// LS Electric XG5000 project: baraka_plc
// PLC NewPLC
// module base 0 slot 0: Input/Output Module:XBC-DR10E (DC 24V INPUT 6points/RELAY OUTPUT 4points)

PROGRAM Program (task: Scan Program)

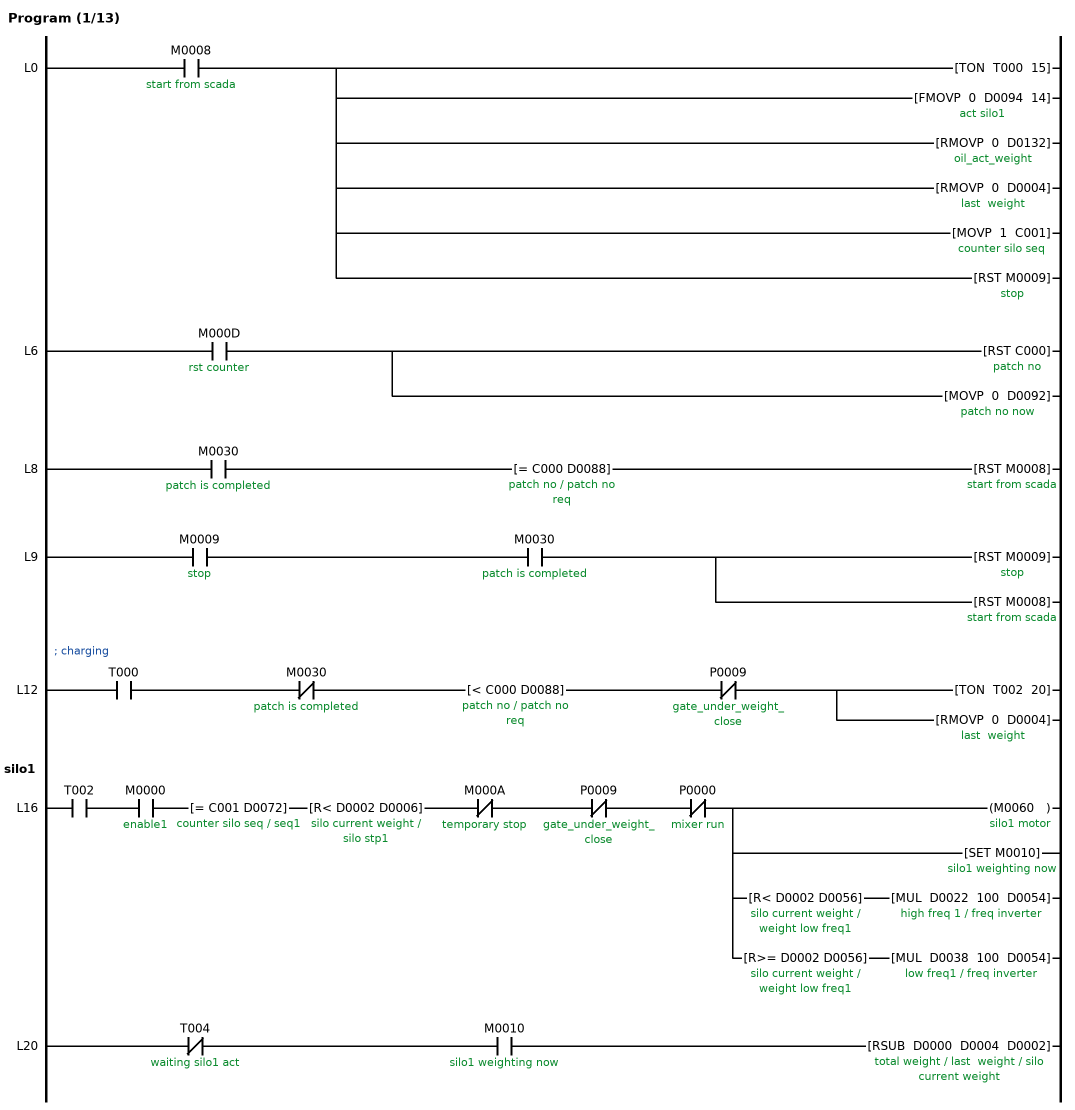
; L0
LOAD      M0008	// start from scada
TON       T000 15
FMOVP     0 D0094 14	// act silo1
RMOVP     0 D0132	// oil_act_weight
RMOVP     0 D0004	// last  weight
MOVP      1 C001	// counter silo seq
RST       M0009	// stop
; L6
LOAD      M000D	// rst counter
RST       C000	// patch no
MOVP      0 D0092	// patch no now
; L8
LOAD      M0030	// patch is completed
AND=      C000 D0088	// patch no / patch no req
RST       M0008	// start from scada
; L9
LOAD      M0009	// stop
AND       M0030	// patch is completed
RST       M0009	// stop
RST       M0008	// start from scada
// charging
; L12
LOAD      T000
AND NOT   M0030	// patch is completed
AND<      C000 D0088	// patch no / patch no req
AND NOT   P0009	// gate_under_weight_close
TON       T002 20
RMOVP     0 D0004	// last  weight
silo1:
; L16
LOAD      T002
AND       M0000	// enable1
AND=      C001 D0072	// counter silo seq / seq1
ANDR<     D0002 D0006	// silo current weight / silo stp1
AND NOT   M000A	// temporary stop
AND NOT   P0009	// gate_under_weight_close
AND NOT   P0000	// mixer run
OUT       M0060	// silo1 motor
SET       M0010	// silo1 weighting now
MPUSH
ANDR<     D0002 D0056	// silo current weight / weight low freq1
MUL       D0022 100 D0054	// high freq 1 / freq inverter
MPOP
ANDR>=    D0002 D0056	// silo current weight / weight low freq1
MUL       D0038 100 D0054	// low freq1 / freq inverter
; L20
LOAD NOT  T004	// waiting silo1 act
AND       M0010	// silo1 weighting now
RSUB      D0000 D0004 D0002	// total weight / last  weight / silo current weight

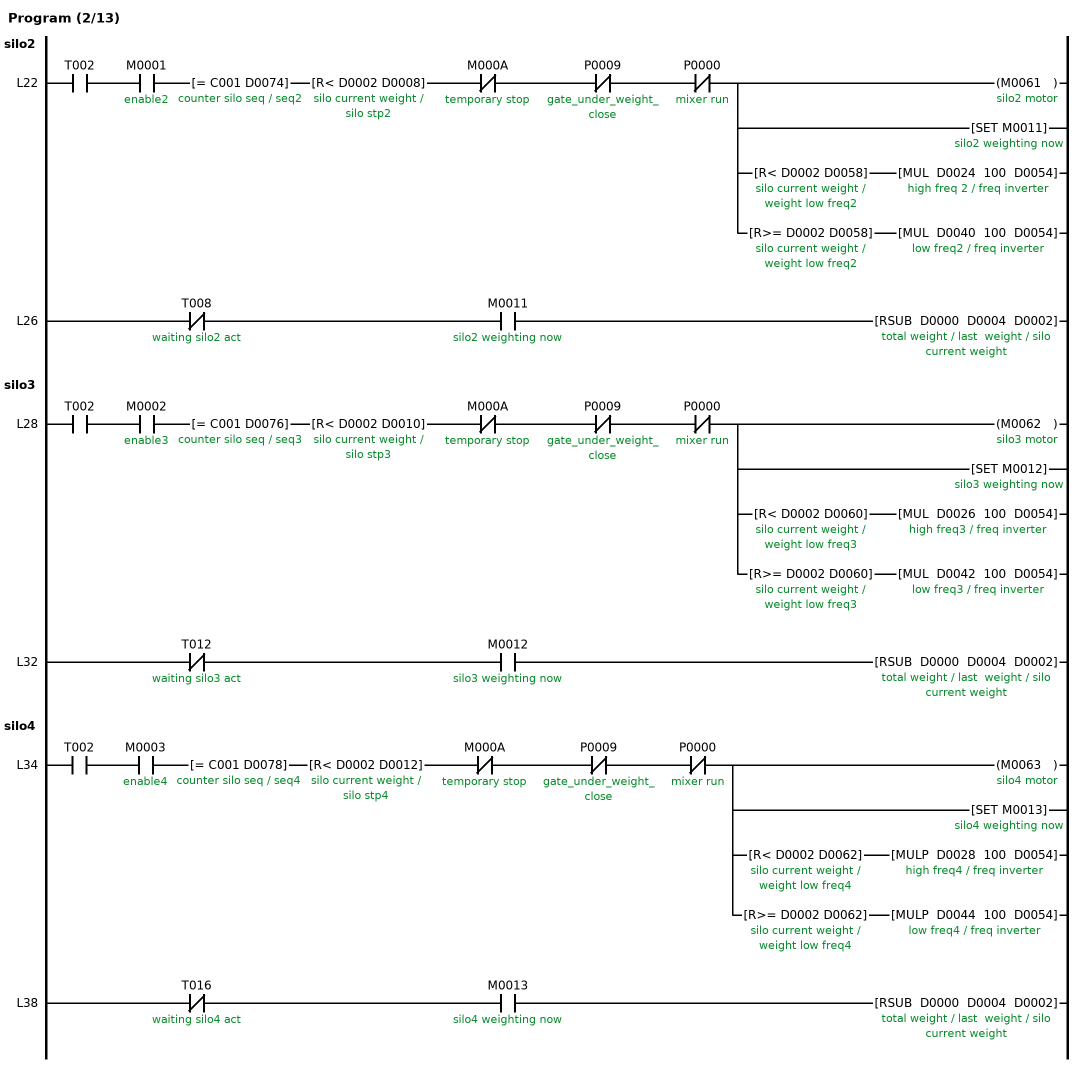
silo2:
; L22
LOAD      T002
AND       M0001	// enable2
AND=      C001 D0074	// counter silo seq / seq2
ANDR<     D0002 D0008	// silo current weight / silo stp2
AND NOT   M000A	// temporary stop
AND NOT   P0009	// gate_under_weight_close
AND NOT   P0000	// mixer run
OUT       M0061	// silo2 motor
SET       M0011	// silo2 weighting now
MPUSH
ANDR<     D0002 D0058	// silo current weight / weight low freq2
MUL       D0024 100 D0054	// high freq 2 / freq inverter
MPOP
ANDR>=    D0002 D0058	// silo current weight / weight low freq2
MUL       D0040 100 D0054	// low freq2 / freq inverter
; L26
LOAD NOT  T008	// waiting silo2 act
AND       M0011	// silo2 weighting now
RSUB      D0000 D0004 D0002	// total weight / last  weight / silo current weight
silo3:
; L28
LOAD      T002
AND       M0002	// enable3
AND=      C001 D0076	// counter silo seq / seq3
ANDR<     D0002 D0010	// silo current weight / silo stp3
AND NOT   M000A	// temporary stop
AND NOT   P0009	// gate_under_weight_close
AND NOT   P0000	// mixer run
OUT       M0062	// silo3 motor
SET       M0012	// silo3 weighting now
MPUSH
ANDR<     D0002 D0060	// silo current weight / weight low freq3
MUL       D0026 100 D0054	// high freq3 / freq inverter
MPOP
ANDR>=    D0002 D0060	// silo current weight / weight low freq3
MUL       D0042 100 D0054	// low freq3 / freq inverter
; L32
LOAD NOT  T012	// waiting silo3 act
AND       M0012	// silo3 weighting now
RSUB      D0000 D0004 D0002	// total weight / last  weight / silo current weight
silo4:
; L34
LOAD      T002
AND       M0003	// enable4
AND=      C001 D0078	// counter silo seq / seq4
ANDR<     D0002 D0012	// silo current weight / silo stp4
AND NOT   M000A	// temporary stop
AND NOT   P0009	// gate_under_weight_close
AND NOT   P0000	// mixer run
OUT       M0063	// silo4 motor
SET       M0013	// silo4 weighting now
MPUSH
ANDR<     D0002 D0062	// silo current weight / weight low freq4
MULP      D0028 100 D0054	// high freq4 / freq inverter
MPOP
ANDR>=    D0002 D0062	// silo current weight / weight low freq4
MULP      D0044 100 D0054	// low freq4 / freq inverter
; L38
LOAD NOT  T016	// waiting silo4 act
AND       M0013	// silo4 weighting now
RSUB      D0000 D0004 D0002	// total weight / last  weight / silo current weight

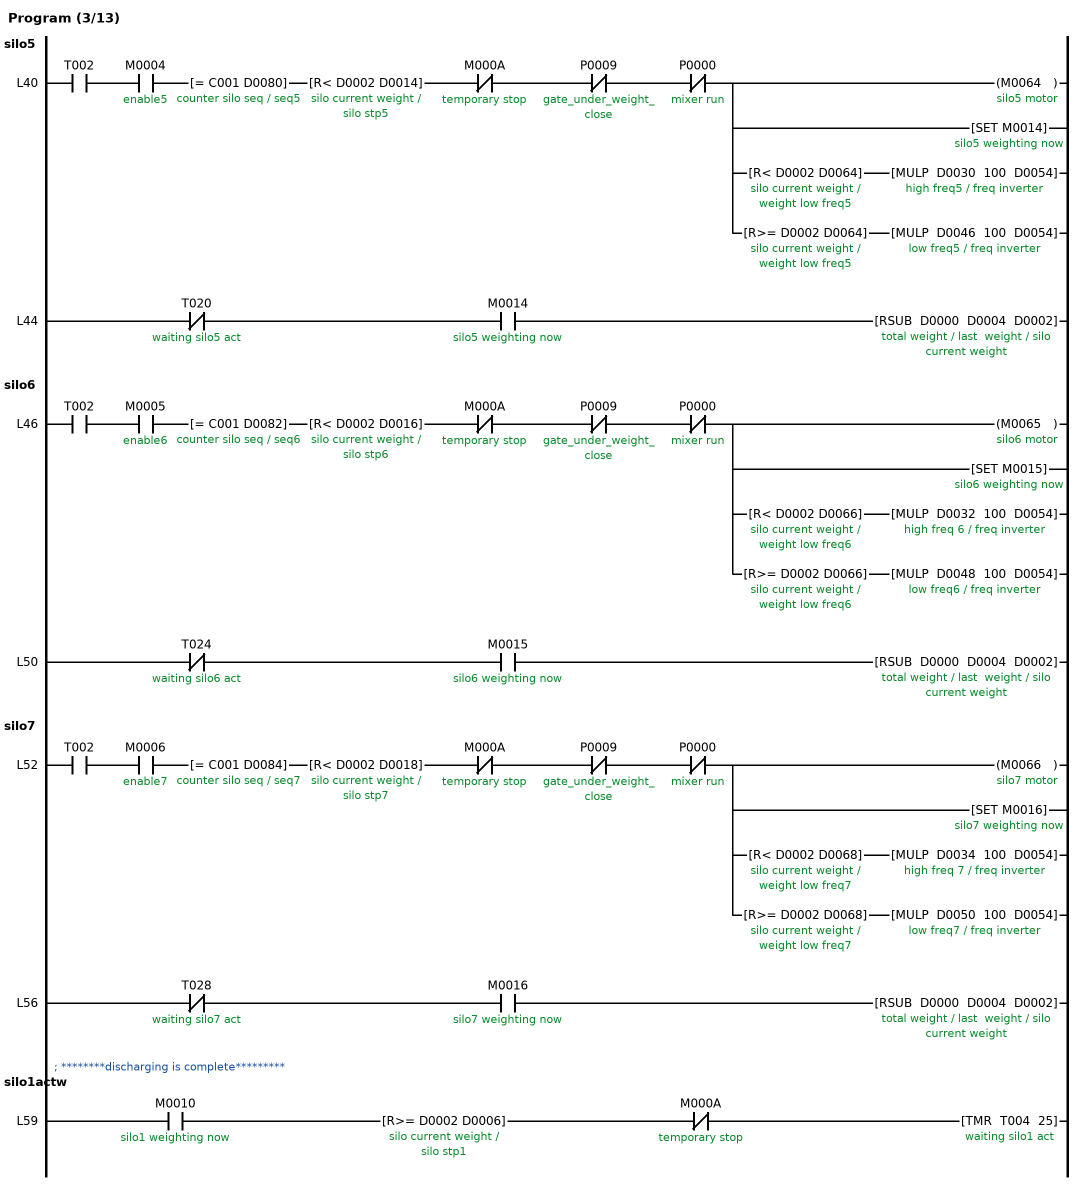
silo5:
; L40
LOAD      T002
AND       M0004	// enable5
AND=      C001 D0080	// counter silo seq / seq5
ANDR<     D0002 D0014	// silo current weight / silo stp5
AND NOT   M000A	// temporary stop
AND NOT   P0009	// gate_under_weight_close
AND NOT   P0000	// mixer run
OUT       M0064	// silo5 motor
SET       M0014	// silo5 weighting now
MPUSH
ANDR<     D0002 D0064	// silo current weight / weight low freq5
MULP      D0030 100 D0054	// high freq5 / freq inverter
MPOP
ANDR>=    D0002 D0064	// silo current weight / weight low freq5
MULP      D0046 100 D0054	// low freq5 / freq inverter
; L44
LOAD NOT  T020	// waiting silo5 act
AND       M0014	// silo5 weighting now
RSUB      D0000 D0004 D0002	// total weight / last  weight / silo current weight
silo6:
; L46
LOAD      T002
AND       M0005	// enable6
AND=      C001 D0082	// counter silo seq / seq6
ANDR<     D0002 D0016	// silo current weight / silo stp6
AND NOT   M000A	// temporary stop
AND NOT   P0009	// gate_under_weight_close
AND NOT   P0000	// mixer run
OUT       M0065	// silo6 motor
SET       M0015	// silo6 weighting now
MPUSH
ANDR<     D0002 D0066	// silo current weight / weight low freq6
MULP      D0032 100 D0054	// high freq 6 / freq inverter
MPOP
ANDR>=    D0002 D0066	// silo current weight / weight low freq6
MULP      D0048 100 D0054	// low freq6 / freq inverter
; L50
LOAD NOT  T024	// waiting silo6 act
AND       M0015	// silo6 weighting now
RSUB      D0000 D0004 D0002	// total weight / last  weight / silo current weight
silo7:
; L52
LOAD      T002
AND       M0006	// enable7
AND=      C001 D0084	// counter silo seq / seq7
ANDR<     D0002 D0018	// silo current weight / silo stp7
AND NOT   M000A	// temporary stop
AND NOT   P0009	// gate_under_weight_close
AND NOT   P0000	// mixer run
OUT       M0066	// silo7 motor
SET       M0016	// silo7 weighting now
MPUSH
ANDR<     D0002 D0068	// silo current weight / weight low freq7
MULP      D0034 100 D0054	// high freq 7 / freq inverter
MPOP
ANDR>=    D0002 D0068	// silo current weight / weight low freq7
MULP      D0050 100 D0054	// low freq7 / freq inverter
; L56
LOAD NOT  T028	// waiting silo7 act
AND       M0016	// silo7 weighting now
RSUB      D0000 D0004 D0002	// total weight / last  weight / silo current weight
// ********discharging is complete*********
silo1actw:
; L59
LOAD      M0010	// silo1 weighting now
ANDR>=    D0002 D0006	// silo current weight / silo stp1
AND NOT   M000A	// temporary stop
TMR       T004 25	// waiting silo1 act

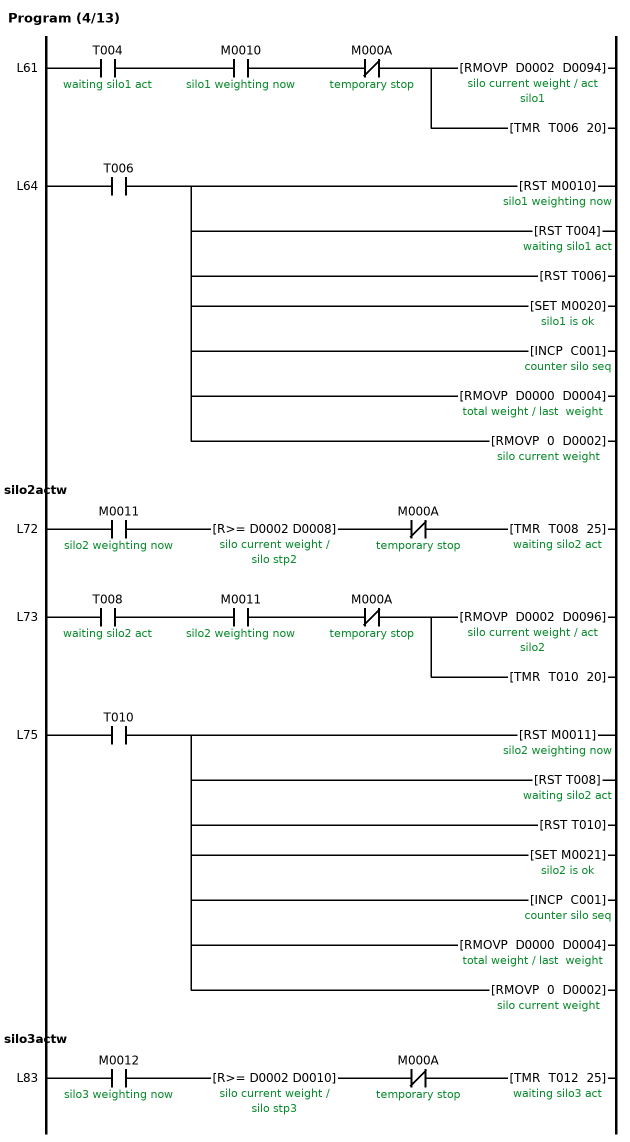
; L61
LOAD      T004	// waiting silo1 act
AND       M0010	// silo1 weighting now
AND NOT   M000A	// temporary stop
RMOVP     D0002 D0094	// silo current weight / act silo1
TMR       T006 20
; L64
LOAD      T006
RST       M0010	// silo1 weighting now
RST       T004	// waiting silo1 act
RST       T006
SET       M0020	// silo1 is ok
INCP      C001	// counter silo seq
RMOVP     D0000 D0004	// total weight / last  weight
RMOVP     0 D0002	// silo current weight
silo2actw:
; L72
LOAD      M0011	// silo2 weighting now
ANDR>=    D0002 D0008	// silo current weight / silo stp2
AND NOT   M000A	// temporary stop
TMR       T008 25	// waiting silo2 act
; L73
LOAD      T008	// waiting silo2 act
AND       M0011	// silo2 weighting now
AND NOT   M000A	// temporary stop
RMOVP     D0002 D0096	// silo current weight / act silo2
TMR       T010 20
; L75
LOAD      T010
RST       M0011	// silo2 weighting now
RST       T008	// waiting silo2 act
RST       T010
SET       M0021	// silo2 is ok
INCP      C001	// counter silo seq
RMOVP     D0000 D0004	// total weight / last  weight
RMOVP     0 D0002	// silo current weight
silo3actw:
; L83
LOAD      M0012	// silo3 weighting now
ANDR>=    D0002 D0010	// silo current weight / silo stp3
AND NOT   M000A	// temporary stop
TMR       T012 25	// waiting silo3 act

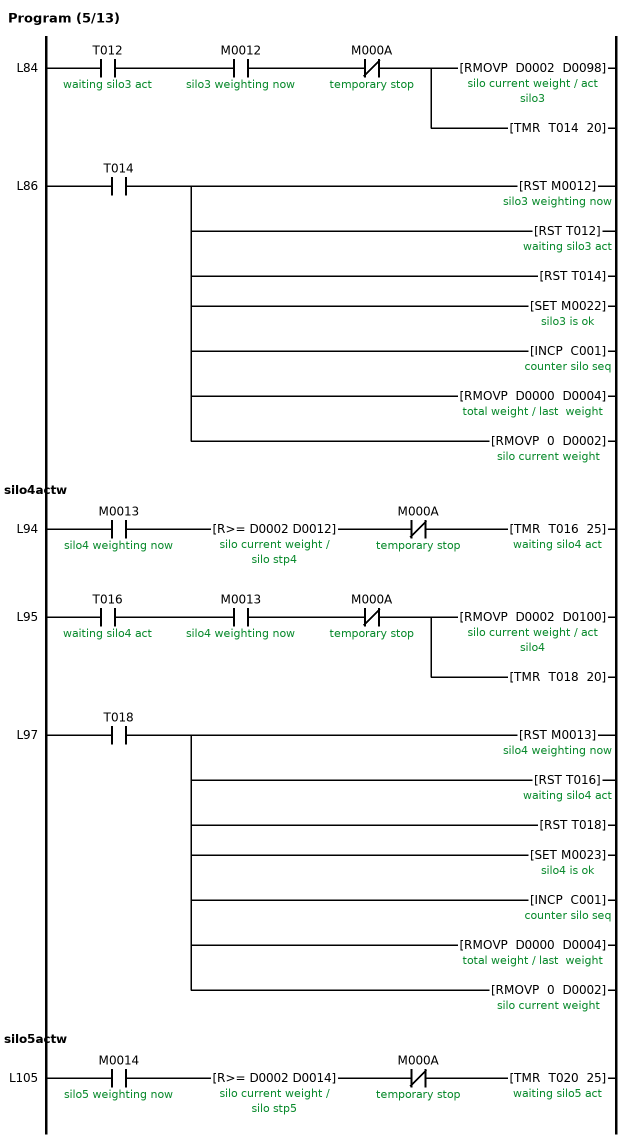
; L84
LOAD      T012	// waiting silo3 act
AND       M0012	// silo3 weighting now
AND NOT   M000A	// temporary stop
RMOVP     D0002 D0098	// silo current weight / act silo3
TMR       T014 20
; L86
LOAD      T014
RST       M0012	// silo3 weighting now
RST       T012	// waiting silo3 act
RST       T014
SET       M0022	// silo3 is ok
INCP      C001	// counter silo seq
RMOVP     D0000 D0004	// total weight / last  weight
RMOVP     0 D0002	// silo current weight
silo4actw:
; L94
LOAD      M0013	// silo4 weighting now
ANDR>=    D0002 D0012	// silo current weight / silo stp4
AND NOT   M000A	// temporary stop
TMR       T016 25	// waiting silo4 act
; L95
LOAD      T016	// waiting silo4 act
AND       M0013	// silo4 weighting now
AND NOT   M000A	// temporary stop
RMOVP     D0002 D0100	// silo current weight / act silo4
TMR       T018 20
; L97
LOAD      T018
RST       M0013	// silo4 weighting now
RST       T016	// waiting silo4 act
RST       T018
SET       M0023	// silo4 is ok
INCP      C001	// counter silo seq
RMOVP     D0000 D0004	// total weight / last  weight
RMOVP     0 D0002	// silo current weight
silo5actw:
; L105
LOAD      M0014	// silo5 weighting now
ANDR>=    D0002 D0014	// silo current weight / silo stp5
AND NOT   M000A	// temporary stop
TMR       T020 25	// waiting silo5 act

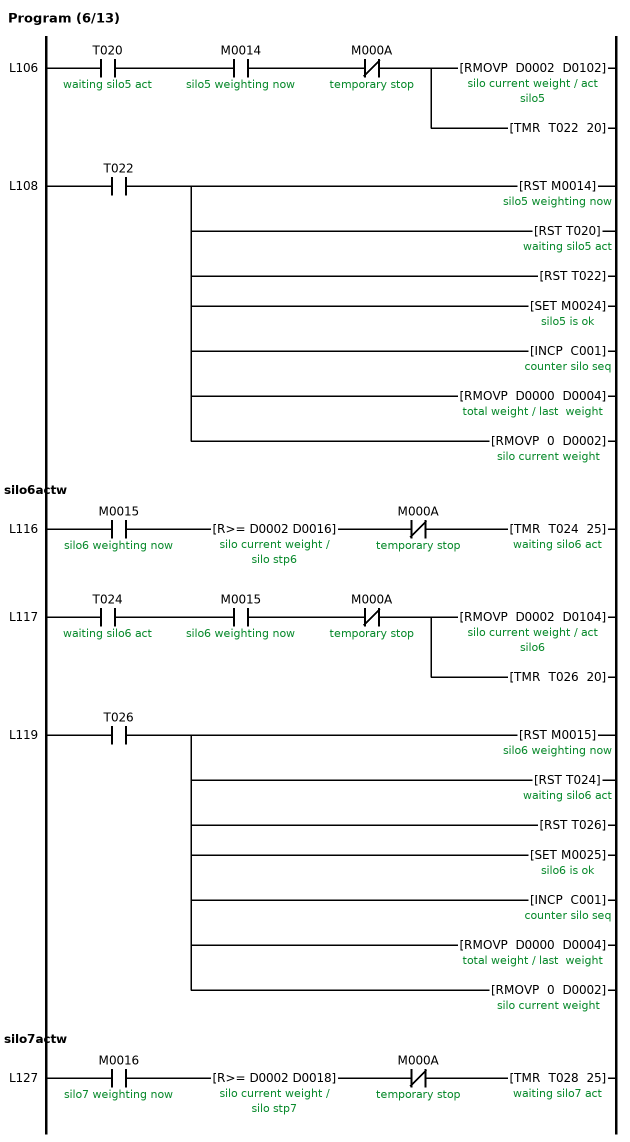
; L106
LOAD      T020	// waiting silo5 act
AND       M0014	// silo5 weighting now
AND NOT   M000A	// temporary stop
RMOVP     D0002 D0102	// silo current weight / act silo5
TMR       T022 20
; L108
LOAD      T022
RST       M0014	// silo5 weighting now
RST       T020	// waiting silo5 act
RST       T022
SET       M0024	// silo5 is ok
INCP      C001	// counter silo seq
RMOVP     D0000 D0004	// total weight / last  weight
RMOVP     0 D0002	// silo current weight
silo6actw:
; L116
LOAD      M0015	// silo6 weighting now
ANDR>=    D0002 D0016	// silo current weight / silo stp6
AND NOT   M000A	// temporary stop
TMR       T024 25	// waiting silo6 act
; L117
LOAD      T024	// waiting silo6 act
AND       M0015	// silo6 weighting now
AND NOT   M000A	// temporary stop
RMOVP     D0002 D0104	// silo current weight / act silo6
TMR       T026 20
; L119
LOAD      T026
RST       M0015	// silo6 weighting now
RST       T024	// waiting silo6 act
RST       T026
SET       M0025	// silo6 is ok
INCP      C001	// counter silo seq
RMOVP     D0000 D0004	// total weight / last  weight
RMOVP     0 D0002	// silo current weight
silo7actw:
; L127
LOAD      M0016	// silo7 weighting now
ANDR>=    D0002 D0018	// silo current weight / silo stp7
AND NOT   M000A	// temporary stop
TMR       T028 25	// waiting silo7 act

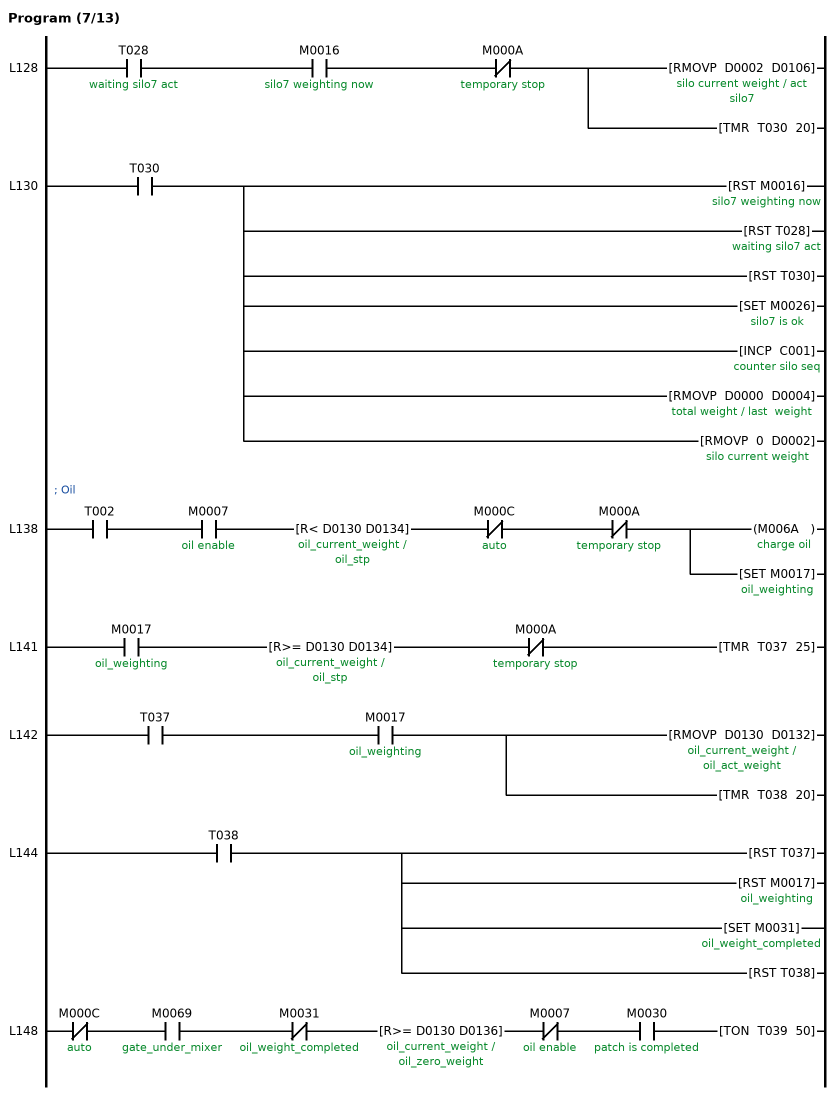
; L128
LOAD      T028	// waiting silo7 act
AND       M0016	// silo7 weighting now
AND NOT   M000A	// temporary stop
RMOVP     D0002 D0106	// silo current weight / act silo7
TMR       T030 20
; L130
LOAD      T030
RST       M0016	// silo7 weighting now
RST       T028	// waiting silo7 act
RST       T030
SET       M0026	// silo7 is ok
INCP      C001	// counter silo seq
RMOVP     D0000 D0004	// total weight / last  weight
RMOVP     0 D0002	// silo current weight
// Oil
; L138
LOAD      T002
AND       M0007	// oil enable
ANDR<     D0130 D0134	// oil_current_weight / oil_stp
AND NOT   M000C	// auto
AND NOT   M000A	// temporary stop
OUT       M006A	// charge oil
SET       M0017	// oil_weighting
; L141
LOAD      M0017	// oil_weighting
ANDR>=    D0130 D0134	// oil_current_weight / oil_stp
AND NOT   M000A	// temporary stop
TMR       T037 25
; L142
LOAD      T037
AND       M0017	// oil_weighting
RMOVP     D0130 D0132	// oil_current_weight / oil_act_weight
TMR       T038 20
; L144
LOAD      T038
RST       T037
RST       M0017	// oil_weighting
SET       M0031	// oil_weight_completed
RST       T038
; L148
LOAD NOT  M000C	// auto
AND       M0069	// gate_under_mixer
AND NOT   M0031	// oil_weight_completed
ANDR>=    D0130 D0136	// oil_current_weight / oil_zero_weight
AND NOT   M0007	// oil enable
AND       M0030	// patch is completed
TON       T039 50

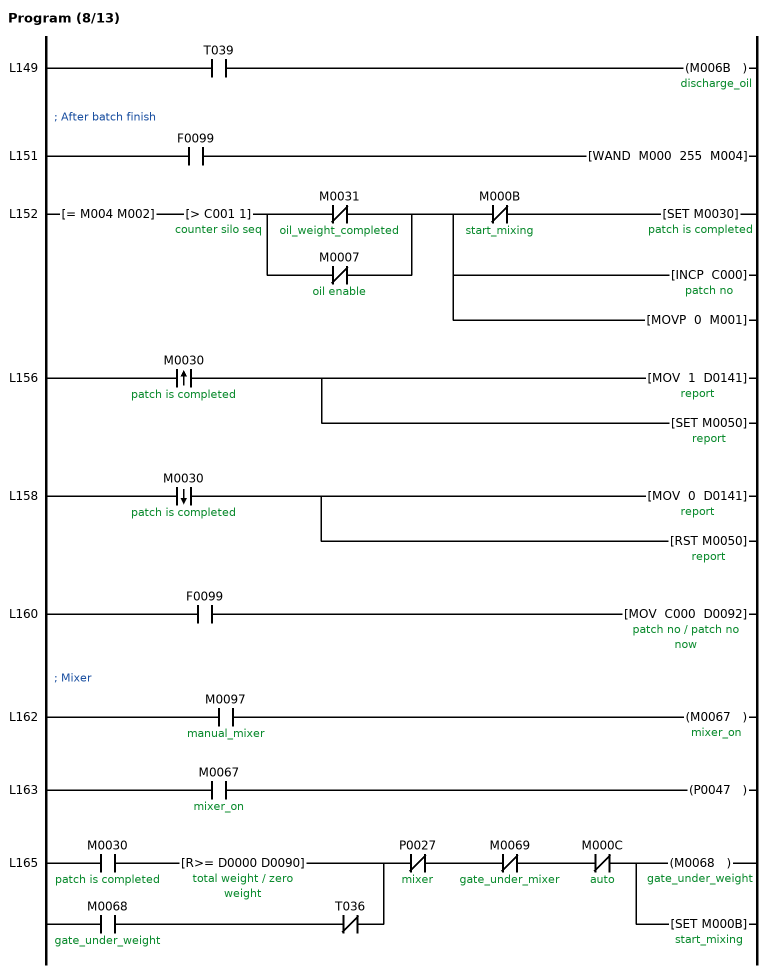
; L149
LOAD      T039
OUT       M006B	// discharge_oil
// After batch finish
; L151
LOAD      F0099
WAND      M000 255 M004
; L152
LOAD=     M004 M002
AND>      C001 1	// counter silo seq
LOAD NOT  M0031	// oil_weight_completed
OR NOT    M0007	// oil enable
AND LOAD
MPUSH
AND NOT   M000B	// start_mixing
SET       M0030	// patch is completed
MPOP
INCP      C000	// patch no
MOVP      0 M001
; L156
LOADP     M0030	// patch is completed
MOV       1 D0141	// report
SET       M0050	// report
; L158
LOADN     M0030	// patch is completed
MOV       0 D0141	// report
RST       M0050	// report
; L160
LOAD      F0099
MOV       C000 D0092	// patch no / patch no now
// Mixer
; L162
LOAD      M0097	// manual_mixer
OUT       M0067	// mixer_on
; L163
LOAD      M0067	// mixer_on
OUT       P0047
; L165
LOAD      M0030	// patch is completed
ANDR>=    D0000 D0090	// total weight / zero weight
LOAD      M0068	// gate_under_weight
AND NOT   T036
OR LOAD
AND NOT   P0027	// mixer
AND NOT   M0069	// gate_under_mixer
AND NOT   M000C	// auto
OUT       M0068	// gate_under_weight
SET       M000B	// start_mixing

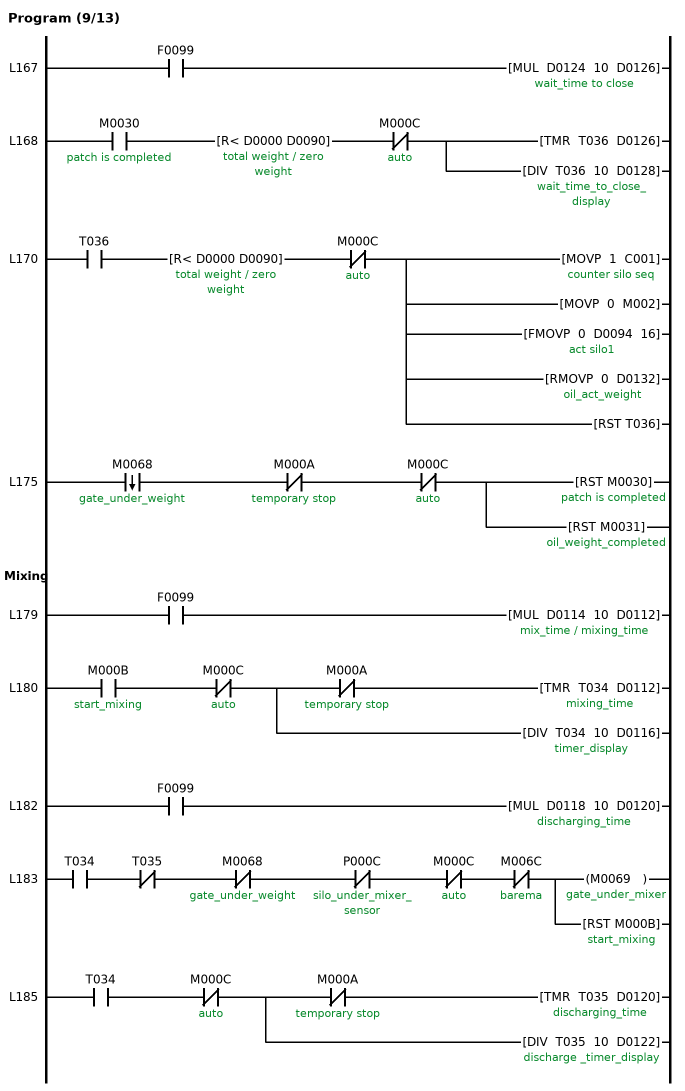
; L167
LOAD      F0099
MUL       D0124 10 D0126	// wait_time to close
; L168
LOAD      M0030	// patch is completed
ANDR<     D0000 D0090	// total weight / zero weight
AND NOT   M000C	// auto
TMR       T036 D0126
DIV       T036 10 D0128	// wait_time_to_close_display
; L170
LOAD      T036
ANDR<     D0000 D0090	// total weight / zero weight
AND NOT   M000C	// auto
MOVP      1 C001	// counter silo seq
MOVP      0 M002
FMOVP     0 D0094 16	// act silo1
RMOVP     0 D0132	// oil_act_weight
RST       T036
; L175
LOADN     M0068	// gate_under_weight
AND NOT   M000A	// temporary stop
AND NOT   M000C	// auto
RST       M0030	// patch is completed
RST       M0031	// oil_weight_completed
Mixing:
; L179
LOAD      F0099
MUL       D0114 10 D0112	// mix_time / mixing_time
; L180
LOAD      M000B	// start_mixing
AND NOT   M000C	// auto
MPUSH
AND NOT   M000A	// temporary stop
TMR       T034 D0112	// mixing_time
MPOP
DIV       T034 10 D0116	// timer_display
; L182
LOAD      F0099
MUL       D0118 10 D0120	// discharging_time
; L183
LOAD      T034
AND NOT   T035
AND NOT   M0068	// gate_under_weight
AND NOT   P000C	// silo_under_mixer_sensor
AND NOT   M000C	// auto
AND NOT   M006C	// barema
OUT       M0069	// gate_under_mixer
RST       M000B	// start_mixing
; L185
LOAD      T034
AND NOT   M000C	// auto
MPUSH
AND NOT   M000A	// temporary stop
TMR       T035 D0120	// discharging_time
MPOP
DIV       T035 10 D0122	// discharge _timer_display

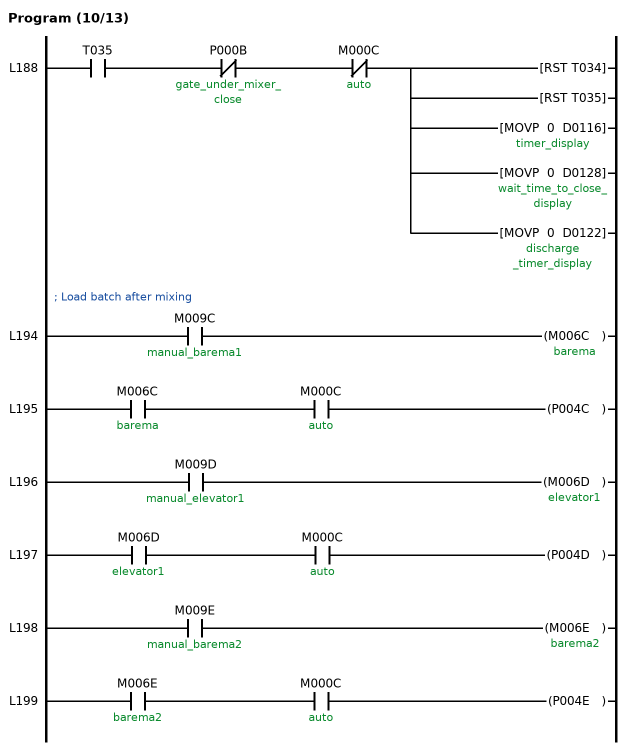
; L188
LOAD      T035
AND NOT   P000B	// gate_under_mixer_close
AND NOT   M000C	// auto
RST       T034
RST       T035
MOVP      0 D0116	// timer_display
MOVP      0 D0128	// wait_time_to_close_display
MOVP      0 D0122	// discharge _timer_display
// Load batch after mixing
; L194
LOAD      M009C	// manual_barema1
OUT       M006C	// barema
; L195
LOAD      M006C	// barema
AND       M000C	// auto
OUT       P004C
; L196
LOAD      M009D	// manual_elevator1
OUT       M006D	// elevator1
; L197
LOAD      M006D	// elevator1
AND       M000C	// auto
OUT       P004D
; L198
LOAD      M009E	// manual_barema2
OUT       M006E	// barema2
; L199
LOAD      M006E	// barema2
AND       M000C	// auto
OUT       P004E

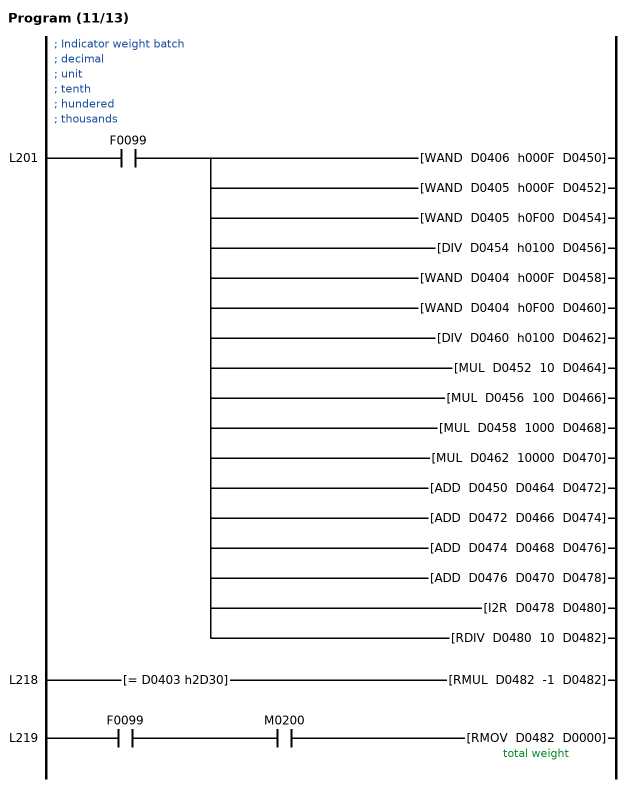
// Indicator weight batch
; L201
LOAD      F0099
WAND      D0406 h000F D0450
WAND      D0405 h000F D0452
WAND      D0405 h0F00 D0454
DIV       D0454 h0100 D0456
WAND      D0404 h000F D0458
WAND      D0404 h0F00 D0460
DIV       D0460 h0100 D0462
MUL       D0452 10 D0464
MUL       D0456 100 D0466
MUL       D0458 1000 D0468
MUL       D0462 10000 D0470
ADD       D0450 D0464 D0472
ADD       D0472 D0466 D0474
ADD       D0474 D0468 D0476
ADD       D0476 D0470 D0478
I2R       D0478 D0480
RDIV      D0480 10 D0482
// output comment: decimal
// output comment: unit
// output comment: tenth
// output comment: hundered
// output comment: thousands
; L218
LOAD=     D0403 h2D30
RMUL      D0482 -1 D0482
; L219
LOAD      F0099
AND       M0200
RMOV      D0482 D0000	// total weight

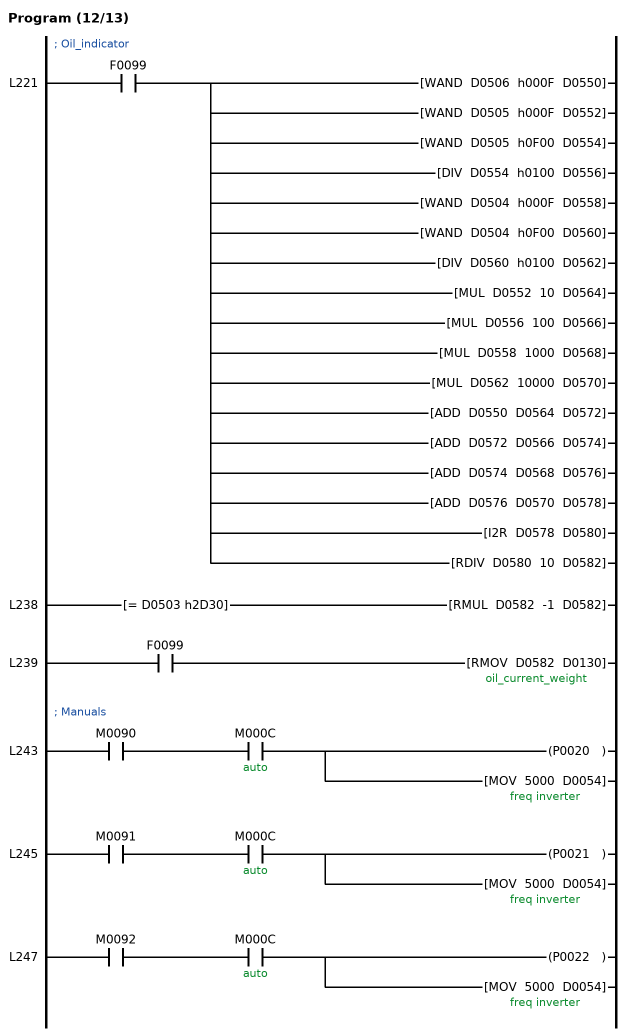
// Oil_indicator
; L221
LOAD      F0099
WAND      D0506 h000F D0550
WAND      D0505 h000F D0552
WAND      D0505 h0F00 D0554
DIV       D0554 h0100 D0556
WAND      D0504 h000F D0558
WAND      D0504 h0F00 D0560
DIV       D0560 h0100 D0562
MUL       D0552 10 D0564
MUL       D0556 100 D0566
MUL       D0558 1000 D0568
MUL       D0562 10000 D0570
ADD       D0550 D0564 D0572
ADD       D0572 D0566 D0574
ADD       D0574 D0568 D0576
ADD       D0576 D0570 D0578
I2R       D0578 D0580
RDIV      D0580 10 D0582
; L238
LOAD=     D0503 h2D30
RMUL      D0582 -1 D0582
; L239
LOAD      F0099
RMOV      D0582 D0130	// oil_current_weight
// Manuals
; L243
LOAD      M0090
AND       M000C	// auto
OUT       P0020
MOV       5000 D0054	// freq inverter
; L245
LOAD      M0091
AND       M000C	// auto
OUT       P0021
MOV       5000 D0054	// freq inverter
; L247
LOAD      M0092
AND       M000C	// auto
OUT       P0022
MOV       5000 D0054	// freq inverter

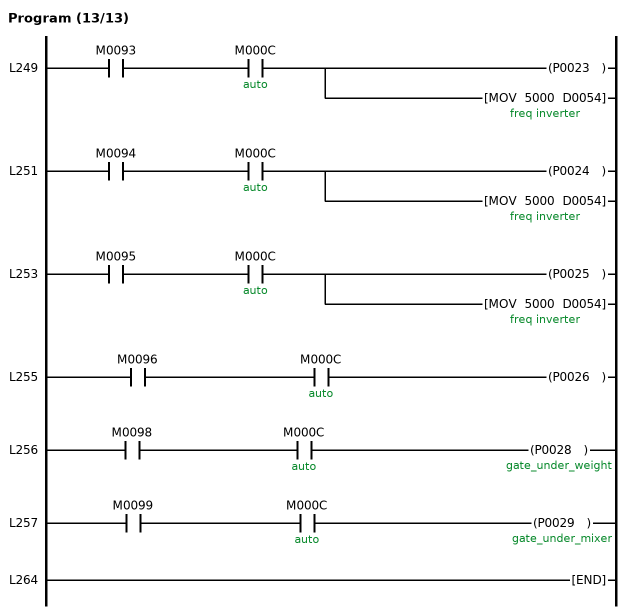
; L249
LOAD      M0093
AND       M000C	// auto
OUT       P0023
MOV       5000 D0054	// freq inverter
; L251
LOAD      M0094
AND       M000C	// auto
OUT       P0024
MOV       5000 D0054	// freq inverter
; L253
LOAD      M0095
AND       M000C	// auto
OUT       P0025
MOV       5000 D0054	// freq inverter
; L255
LOAD      M0096
AND       M000C	// auto
OUT       P0026
; L256
LOAD      M0098
AND       M000C	// auto
OUT       P0028	// gate_under_weight
; L257
LOAD      M0099
AND       M000C	// auto
OUT       P0029	// gate_under_mixer
; L264
END

PROGRAM inverter&outputs&inputs (task: Scan Program)

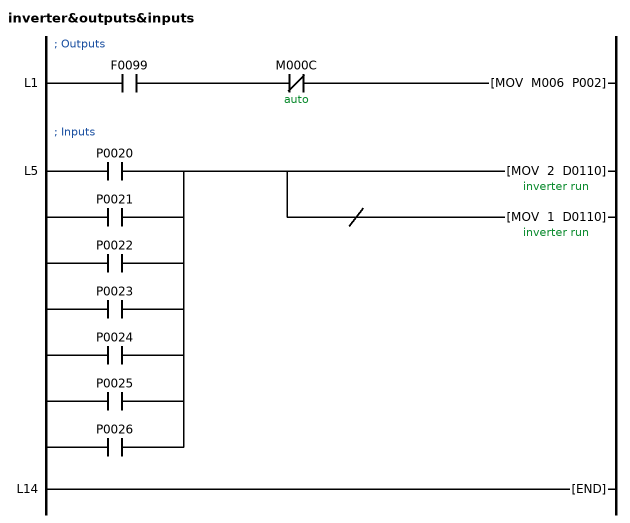
// Outputs
; L1
LOAD      F0099
AND NOT   M000C	// auto
MOV       M006 P002
// Inputs
; L5
LOAD      P0020
OR        P0021
OR        P0022
OR        P0023
OR        P0024
OR        P0025
OR        P0026
MOV       2 D0110	// inverter run
NOT
MOV       1 D0110	// inverter run
; L14
END

VARIABLES AND COMMENTS (devices not used above)
D00020	WORD	silo stp 8
D00036	WORD	high freq 8
D00052	WORD	low freq8
D00070	WORD	weight low freq8
D00086	WORD	seq8
D00108	WORD	act silo8
T0032	BIT/WORD	waiting silo8 act
M00027	BIT	silo8 is ok
P00008	BIT	gate_under_weight_open
P0000A	BIT	gate_under_mixer_open
P0002A	BIT	barema2
P0002D	BIT	elevator1
P0002E	BIT	barema2
D00140	WORD	oil_stp
P0002C	BIT	barema
M00032	BIT	patch enter